// TwinCAT 3 PLC project Machine_Control
// ProgramVersion: 3.1.4024.0
// libraries:
//   Tc2_Drive, * (Beckhoff Automation GmbH)
//   Tc2_EtherCAT, * (Beckhoff Automation GmbH)
//   Tc2_Standard, * (Beckhoff Automation GmbH)
//   Tc2_System, * (Beckhoff Automation GmbH)
//   Tc3_Module, * (Beckhoff Automation GmbH)
// project tree:
//   GVLs/ GVL_Exceptions.TcGVL, GVL_STRUCT.TcGVL, GVL_VAR.TcGVL
//   / PlcTask.TcTTO
//   POUs/ F_SaveExceptionCode.TcPOU, Motors_Speed_IO.TcPOU, Motor_Speed_PID.TcPOU, Safeties_Product_Feed.TcPOU, SpeedControl_SIM.TcPOU, MAIN.TcPOU
// real-time tasks:
//   TASK PlcTask: cycle T#10ms, priority 20, ADS port 350
// I/O:
//   DEVICE Device 1 (EtherCAT Simulation), AmsNetId 192.168.0.15.2.1

CONFIGURATION Machine_Control
    RESOURCE PLC ON TwinCAT3
        TASK PlcTask(INTERVAL := T#10ms, PRIORITY := 20);
        PROGRAM MAIN WITH PlcTask : MAIN;
    END_RESOURCE
END_CONFIGURATION

// ---- GVLs/GVL_Exceptions.TcGVL
{attribute 'qualified_only'}
VAR_GLOBAL CONSTANT
	
	cMaxExc : UINT := 10;	

END_VAR

VAR_GLOBAL
	
	nExcIndex : UINT;
	aExceptionHistory : ARRAY[0..cMaxExc] OF __SYSTEM.ExceptionCode;

END_VAR

// ---- GVLs/GVL_STRUCT.TcGVL
{attribute 'qualified_only'}
VAR_GLOBAL

END_VAR

TYPE 
ST_DriveRef 	:
STRUCT
	
	sNetId		: T_AmsNetId;
	nSlaveAddr	: UINT	:= GVL_VAR.uiSlaveAddr;
	nDriveNo 	: BYTE	:= GVL_VAR.nDriveNum;
	nDriveType	: BYTE	:= GVL_VAR.nDriveType;
	
END_STRUCT
END_TYPE

// ---- GVLs/GVL_VAR.TcGVL
{attribute 'qualified_only'}
VAR_GLOBAL
	
	//integer variables
	//The values of the rotary encoders are stored into these variables
	diMotorEncoder1 	 	: INT;
	diMotorEncoder2 	 	: INT;
	diMotorEncoder3 	 	: INT;
	diMotorEncoder4 	 	: INT;
	
	//Setting the PPR of the encoders used
	iEncoderPPR 			: INT;
	
	//Speed is calculated after each scan of encoder bits and stored into these variables
	//The values are initialized in order to give the UI something to work with after immediate bootup
	diEncoder1ProdSpeed  	: INT := 0;
	diEncoder2ProdSpeed  	: INT := 0;
	diEncoder3ProdSpeed  	: INT := 0;
	diEncoder4ProdSpeed  	: INT := 0;
	
	//The global speed of motors and overall set-speed
	iMotor1GlobalSpeed   	: INT := 0;
	iMotor2GlobalSpeed   	: INT := 0;
	iMotor3GlobalSpeed   	: INT := 0;
	iMotor4GlobalSpeed   	: INT := 0;
	iSetGlobalSpeed      	: INT := 0;
	iGlobalMinimumFaultSpeed: INT := 40; // This value will be user defined
	
	//An hysteresis is important in order to allow micoradjustments in terms of tolerance
	//The values are initialized in order to give the UI something to work with after immediate bootup
	diEncoder1Hysteresis 	: INT := 0;
	diEncoder2Hysteresis 	: INT := 0;
	diEncoder3Hysteresis 	: INT := 0;
	diEncoder4Hysteresis 	: INT := 0;
	
	//Temperature of gluepot/optical in raw data if anaolgue is used 0-4028 depending on the resolution
	//The values are initialized in order to give the UI something to work with after immediate bootup
	iGlueTemperatureRaw  	: INT := 0;
	iRawBoardOptic1 	 	: INT := 0;
	iRawBoardOptic2  	 	: INT := 0;
	iRawBoardOptic3  	 	: INT := 0;
	iRawBoardOptic4 	 	: INT := 0;
	
	//Amount of times a motor's speed has undergone rectification
	
	iMotor1Rect				: INT;
	iMotor2Rect 			: INT;
	iMotor3Rect 			: INT;
	iMotor4Rect 			: INT;
	
	//Program cutt-off distances
	//This keeps track of material distances if motors lose sync of their speed parameters
	//This will be referenced in conjunction with the "Product Ready" flag which must be set BEFORE product is fed
	//Yet IF product is fed, the precondition must remain true; 
	fProductRun : REAL;
	
	//Motor References VIA EtherCAT Comms methodology
	uiSlaveAddr : UINT;
	nDriveNum	: BYTE;
	nDriveType	: BYTE;
	
	
	//boolean variables
	//As far as feasible the booleans will be initialized
	bStartButton 		 	: BOOL := FALSE;
	bStopButton 		 	: BOOL := FALSE;
	bPauseButton 		 	: BOOL := FALSE;
	//System parameters from the main OS/UI
	bSysParamExec 		 	: BOOL := FALSE;
	bSysParamHold 		 	: BOOL := FALSE;
	bSysParamReset 		 	: BOOL := FALSE;
	bSysParam1 			 	: BOOL := FALSE;
	bSysParam2 			 	: BOOL := FALSE;
	//Some IO information about the motor's state
	bMotor1Running 		 	: BOOL := FALSE;
	bMotor2Running 		 	: BOOL := FALSE;
	bMotor3Running 		 	: BOOL := FALSE;
	bMotor4Running 		 	: BOOL := FALSE;
	//Gluepot Boolean indicators
	bGlueReady 			 	: BOOL := FALSE;
	
	//Output Section for controlling the COILS with boolean values
	bStartMotor1			: BOOL := FALSE;
	bStartMotor2			: BOOL := FALSE;
	bStartMotor3			: BOOL := FALSE;
	bStartMotor4			: BOOL := FALSE;
	bMotorsHaveStarted		: BOOL := FALSE;
	
	//Bolleans for controlling the carious motor's speed:
	//These variables are called again in the PID controller POU Motor_Speed_PID
	bIncreaseSpeed1 		: BOOL := FALSE;
	bDecreaseSpeed1 		: BOOL := FALSE;
	bIncreaseSpeed2 		: BOOL := FALSE;
	bDecreaseSpeed2 		: BOOL := FALSE;
	bIncreaseSpeed3 		: BOOL := FALSE;
	bDecreaseSpeed3 		: BOOL := FALSE;
	bIncreaseSpeed4 		: BOOL := FALSE;
	bDecreaseSpeed4 		: BOOL := FALSE;

//Real variables
	//Temperature of glue pot in degrees celsius
	//The values are initialized in order to give the UI something to work with after immediate bootup
	fGlueTemperature 	 	: REAL := 0.0;
	fBoardOptic1 		 	: REAL := 0.0;
	fBoardOptic2 		 	: REAL := 0.0;
	fBoardOptic3 		 	: REAL := 0.0;
	fBoardOptic4 		 	: REAL := 0.0;
	fMaterialDistanceMeter 	: REAL := 0.0;
	fMotor1Thermal 			: REAL := 0.0;
	fMotor2Thermal 			: REAL := 0.0;
	fMotor3Thermal 			: REAL := 0.0;
	fMotor4Thermal 			: REAL := 0.0;
	
	//REAL values for adjusting the motor speeds after having gone through the Motor_Speed_PID POU
	fMotor1AdjustFactor 	: REAL;
	fMotor2AdjustFactor 	: REAL;
	fMotor3AdjustFactor 	: REAL;
	fMotor4AdjustFactor 	: REAL;
	//REAL value for the hysteresis of the motors speed reference provided to the drives from the Motor_Speed_PID POU
	fMotor1Hysteresis		: REAL;
	fMotor2Hysteresis		: REAL;
	fMotor3Hysteresis		: REAL;
	fMotor4Hysteresis		: REAL;
	
	//This is where the parameters for checking the material highs and lows will be stored
	fParametersOptic1 : REAL;
	fParametersOptic2 : REAL;
	fParametersOptic3 : REAL;
	fParametersOptic4 : REAL;
	
END_VAR

// ---- POUs/MAIN.TcPOU
PROGRAM MAIN
VAR
	bSwitchCtrl		: BOOL := TRUE;
	nRotateUpper	: WORD := 16#8000;
	nRotateLower	: WORD := 16#01;
	
	//Variables for dynamically changing the devices spoken to over EtherCAT
	uiSlaveAddr : UINT;
	nDriveNum	: BYTE;
	nDriveType	: BYTE;
	//For the sake of demonstration I am going to employ a CASE switch for talking to the various drives when initializing...
	iNumDrives	: UINT := 1;
	iDriveType	: UINT := 123;
	
	//Hardware inputs
	bEL1004_CH4 AT%I*	: BOOL;
	stPlcDriveRef AT %I* : ST_PlcDriveRef;
	
	
	nEL2008_value AT%Q*	: BYTE;
	bInit1 : BOOL := FALSE;
	bInit2 : BOOL := FALSE;
	bInit3 : BOOL := FALSE;
	bInit4 : BOOL := FALSE;
	
	//Function Block references
	fbWriteCommandControl 	: FB_SoEWriteCommandControl_ByDriveRef;
	bWriteCommand			: BOOL;	
END_VAR

VAR_INPUT
	//Reference to the drive. The reference to the drive can be linked directly to the PLC in the System Manager. 
	//To do this, an instance of the structure ST_PlcDriveRef must be allocated and the NetID must be converted from the byte array into a string. (Type: ST_DriveRef)
	stDriveRef	: ST_DriveRef;
	//Parameter number to which fbWriteCommandControl refers, e.g. "P_0_IDN + 23" for P-0-0023
	nIdn		: WORD;
	//Indicates, if a command should be prepared (eSoE_CmdControl_Set := 1), executed (eSoE_CmdControl_SetAndEnable := 3) or aborted (eSoE_CmdControl_Cancel := 0).
	eCmdControl	: E_SoE_CmdControl;
	//The function block is enabled via a positive edge at this input
	bExecute	: BOOL;
	//Maximum time (10 s) allowed for the execution of the function block.
	tTimeout	: TIME := DEFAULT_ADS_TIMEOUT;	
END_VAR

VAR_OUTPUT
	//This output is set when the function block is activated, and remains set until a feedback is received.
	bBusy			: BOOL;
	//This output is set after the bBusy output has been reset when an error occurs in the transmission of the command.
	bError			: BOOL;
	//In the case of a set bError output returns the ADS error code of the last executed command.
	iAdsErrId		: UINT;
	//In the case of a set bError output returns the Sercos error of the last executed command.
	iSercosErrId	: UINT;
END_VAR

(*This portion is for dynamic drive communication*)

(*Drives have to be made contact with initially before anything can continue...*)

// A __TRY __CATCH __FINALLY clause will be added for exception handling shortly...

CASE iNumDrives OF //probably the conditional control function I like the most...
//Setting up comms for the motion control needs
	1:	IF NOT bInit1 THEN
		
		//change the Slave address
		uiSlaveAddr := iNumDrives;
		GVL_VAR.uiSlaveAddr := uiSlaveAddr;
		//The structure created for the ST_DriveRef expects a Byte format...hence the conversion of the ints...
		GVL_VAR.nDriveNum	:= INT_TO_BYTE(iNumDrives);
		GVL_VAR.nDriveType	:= INT_TO_BYTE(iDriveType);

		stDriveRef.sNetId		:=	F_CreateAmsNetId(stPlcDriveRef.aNetId);
		//The following values have been preconfigured by the FB
		stDriveRef.nSlaveAddr	:=	GVL_VAR.uiSlaveAddr;
		stDriveRef.nDriveNo		:=	GVL_VAR.nDriveNum;
		stDriveRef.nDriveType	:=	GVL_VAR.nDriveType;
	
		IF (stDriveRef.sNetId <> '') AND (stDriveRef.nSlaveAddr <> 0) THEN
		
		bInit1 := TRUE;//initialization completed
		
		END_IF
	
		END_IF
		
		IF bWriteCommand AND bInit1 THEN
	
			fbWriteCommandControl(
				stDriveRef	:= stDriveRef,
				bExecute	:= TRUE,
				tTimeout	:= DEFAULT_ADS_TIMEOUT,
				nIdn		:= P_0_IDN + 23,
				eCmdControl := eCmdControl
				);
		IF NOT	fbWriteCommandControl.bBusy THEN
			fbWriteCommandControl(stDriveRef := stDriveRef, bExecute := FALSE);
			bWriteCommand := FALSE;			
		END_IF
		
		END_IF
		//increment for the next case...
		iNumDrives := iNumDrives + 1;
		
	2:	IF NOT bInit2 THEN
	
		//change the Slave address
		uiSlaveAddr := iNumDrives;
		GVL_VAR.uiSlaveAddr := uiSlaveAddr;
		//The structure created for the ST_DriveRef expects a Byte format...hence the conversion of the ints...
		GVL_VAR.nDriveNum	:= INT_TO_BYTE(iNumDrives);
		GVL_VAR.nDriveType	:= INT_TO_BYTE(iDriveType);

		stDriveRef.sNetId		:=	F_CreateAmsNetId(stPlcDriveRef.aNetId);
		//The following values have been preconfigured by the FB
		stDriveRef.nSlaveAddr	:=	GVL_VAR.uiSlaveAddr;
		stDriveRef.nDriveNo		:=	GVL_VAR.nDriveNum;
		stDriveRef.nDriveType	:=	GVL_VAR.nDriveType;
	
		IF (stDriveRef.sNetId <> '') AND (stDriveRef.nSlaveAddr <> 0) THEN
		
		bInit2 := TRUE;//initialization completed
		
		END_IF
	
		END_IF
		
		IF bWriteCommand AND bInit2 THEN
	
			fbWriteCommandControl(
				stDriveRef	:= stDriveRef,
				bExecute	:= TRUE,
				tTimeout	:= DEFAULT_ADS_TIMEOUT,
				nIdn		:= P_0_IDN + 23,
				eCmdControl := eCmdControl
				);
		IF NOT	fbWriteCommandControl.bBusy THEN
			fbWriteCommandControl(stDriveRef := stDriveRef, bExecute := FALSE);
			bWriteCommand := FALSE;			
		END_IF
		
		END_IF
		//increment for the next case...
		iNumDrives := iNumDrives + 1;
		
		
	
	3:	IF NOT bInit3 THEN
	
		//change the Slave address
		uiSlaveAddr := iNumDrives;
		GVL_VAR.uiSlaveAddr := uiSlaveAddr;
		//The structure created for the ST_DriveRef expects a Byte format...hence the conversion of the ints...
		GVL_VAR.nDriveNum	:= INT_TO_BYTE(iNumDrives);
		GVL_VAR.nDriveType	:= INT_TO_BYTE(iDriveType);

		stDriveRef.sNetId		:=	F_CreateAmsNetId(stPlcDriveRef.aNetId);
		//The following values have been preconfigured by the FB
		stDriveRef.nSlaveAddr	:=	GVL_VAR.uiSlaveAddr;
		stDriveRef.nDriveNo		:=	GVL_VAR.nDriveNum;
		stDriveRef.nDriveType	:=	GVL_VAR.nDriveType;
	
		IF (stDriveRef.sNetId <> '') AND (stDriveRef.nSlaveAddr <> 0) THEN
		
		bInit3 := TRUE;//initialization completed
		
		END_IF
	
		END_IF
		
		IF bWriteCommand AND bInit3 THEN
	
			fbWriteCommandControl(
				stDriveRef	:= stDriveRef,
				bExecute	:= TRUE,
				tTimeout	:= DEFAULT_ADS_TIMEOUT,
				nIdn		:= P_0_IDN + 23,
				eCmdControl := eCmdControl
				);
		IF NOT	fbWriteCommandControl.bBusy THEN
			fbWriteCommandControl(stDriveRef := stDriveRef, bExecute := FALSE);
			bWriteCommand := FALSE;			
		END_IF
		
		END_IF
		//increment for the next case...
		iNumDrives := iNumDrives + 1;
	
	4:	IF NOT bInit4 THEN
	
		//change the Slave address
		uiSlaveAddr := iNumDrives;
		GVL_VAR.uiSlaveAddr := uiSlaveAddr;
		//The structure created for the ST_DriveRef expects a Byte format...hence the conversion of the ints...
		GVL_VAR.nDriveNum	:= INT_TO_BYTE(iNumDrives);
		GVL_VAR.nDriveType	:= INT_TO_BYTE(iDriveType);

		stDriveRef.sNetId		:=	F_CreateAmsNetId(stPlcDriveRef.aNetId);
		//The following values have been preconfigured by the FB
		stDriveRef.nSlaveAddr	:=	GVL_VAR.uiSlaveAddr;
		stDriveRef.nDriveNo		:=	GVL_VAR.nDriveNum;
		stDriveRef.nDriveType	:=	GVL_VAR.nDriveType;
	
		IF (stDriveRef.sNetId <> '') AND (stDriveRef.nSlaveAddr <> 0) THEN
		
		bInit4 := TRUE;//initialization completed
		
		END_IF
	
		END_IF
		
		IF bWriteCommand AND bInit4 THEN
	
			fbWriteCommandControl(
				stDriveRef	:= stDriveRef,
				bExecute	:= TRUE,
				tTimeout	:= DEFAULT_ADS_TIMEOUT,
				nIdn		:= P_0_IDN + 23,
				eCmdControl := eCmdControl
				);
		IF NOT	fbWriteCommandControl.bBusy THEN
			fbWriteCommandControl(stDriveRef := stDriveRef, bExecute := FALSE);
			bWriteCommand := FALSE;			
		END_IF
		
		END_IF
		//increment for the next case...
		iNumDrives := iNumDrives + 1;
END_CASE




IF bEL1004_CH4 THEN
	IF bSwitchCtrl THEN
		bSwitchCtrl := FALSE;
		nRotateLower := ROL(nRotateUpper, 2);
		nRotateUpper := ROR(nRotateUpper, 2);
		nEL2008_value := WORD_TO_BYTE(nRotateLower OR nRotateUpper);
	END_IF
ELSE
		IF NOT bSwitchCtrl THEN
			bSwitchCtrl := TRUE;
		END_IF
END_IF

END_PROGRAM

// ---- POUs/Motor_Speed_PID.TcPOU
PROGRAM Motor_Speed_PID
VAR
	//Global Variables Assignments
	//Increase or decrease the speed depending on the booleans set by the SpeedControl POU
	//The entire existance of this instance of code assumes no common reference of speed 
	//Basically no servo-motors with trusted speeds are used in the process...
	bIncreaseSpeed1 : BOOL := GVL_VAR.bIncreaseSpeed1;
	bDecreaseSpeed1 : BOOL := GVL_VAR.bDecreaseSpeed1;
	bIncreaseSpeed2 : BOOL := GVL_VAR.bIncreaseSpeed2;
	bDecreaseSpeed2 : BOOL := GVL_VAR.bDecreaseSpeed2;
	bIncreaseSpeed3 : BOOL := GVL_VAR.bIncreaseSpeed3;
	bDecreaseSpeed3 : BOOL := GVL_VAR.bDecreaseSpeed3;
	bIncreaseSpeed4 : BOOL := GVL_VAR.bIncreaseSpeed4;
	bDecreaseSpeed4 : BOOL := GVL_VAR.bDecreaseSpeed4;
	
	//The motor VFD controls have to be referenced here as well... This may be done via some etherCAT comms
	
	//Global speed setting for hte reference of the PID
	iSetGlobalSpeed : INT := GVL_VAR.iSetGlobalSpeed;
	fKp : REAL := 0; //Controller amplification, this is the value sent to the motor controller
	//These are the outputs of the Proportional function to be sent to the drives after encoder references.
	fMotor1AdjustFactor : REAL := GVL_VAR.fMotor1AdjustFactor;
	fMotor2AdjustFactor : REAL := GVL_VAR.fMotor2AdjustFactor;
	fMotor3AdjustFactor : REAL := GVL_VAR.fMotor3AdjustFactor;
	fMotor4AdjustFactor : REAL := GVL_VAR.fMotor4AdjustFactor;
	
	//Reference for the varioous drives' addresses
	//Reference to the drive. The reference to the drive can be linked directly to the PLC in the System Manager.
	//To do this, an instance of the structure ST_PlcDriveRef must be allocated and the 
	//NetID must be converted from the byte array into a string
	
	
END_VAR

//Only allow the activation of the speed control segment of the program if the motors have actually started:

WHILE GVL_VAR.bMotorsHaveStarted DO
	
	//Run through the scans to verify whether or not the logic must start:
	IF bIncreaseSpeed1 OR bDecreaseSpeed1 THEN
	
															//This clause is to keep the motors from going in reverse
		IF GVL_VAR.iMotor1GlobalSpeed < iSetGlobalSpeed AND GVL_VAR.iMotor1GlobalSpeed > 0.0 THEN
		//increase the speed and after making sure the speed doesn't exceed the global set variable for the overall speed
		//determine the factor by which the speed should be increased
		
		//The formula for Proportional control is: P = Kp * (Setpoint - Feedback)
		//Or in this case: GVL_VAR.iMotor1GlobalSpeed := fKp * (GVL_VAR.iSetGlobalSpeed - GVl_VAR.iMotor1GlobalSpeed);
		//So it will look like this (remember this automatically returns a REAL number (Fractional/Decimal)):
		//If you wish to turn a REAL value into an INT value: INT_Value := TRUNC(REAL_Value);
		fMotor1AdjustFactor := fKp * (iSetGlobalSpeed - GVL_VAR.iMotor1GlobalSpeed);	
		//Remember to include a function for keeping the hysteresis in mind.
		GVL_VAR.fMotor1AdjustFactor := fMotor1AdjustFactor - GVL_VAR.fMotor1Hysteresis;
		//increase the speed and after making sure the speed doesn't exceed the global set variable for the overall speed


	
		//Reset the booleans responsible for activating this function
		GVL_VAR.bDecreaseSpeed1 := FALSE;
		GVL_VAR.bIncreaseSpeed1 := FALSE;
		ELSE
		//post a speed reference error
		//Reset the booleans responsible for activating this function
		GVL_VAR.bDecreaseSpeed1 := FALSE;
		GVL_VAR.bIncreaseSpeed1 := FALSE;			
		 
			
		END_IF
		
	END_IF
	
		//Run through the scans to verify whether or not the logic must start:
	IF bIncreaseSpeed2 OR bDecreaseSpeed2 THEN
	
		
		IF GVL_VAR.iMotor1GlobalSpeed < iSetGlobalSpeed AND GVL_VAR.iMotor2GlobalSpeed > 0.0 THEN
		fMotor2AdjustFactor := fKp * (iSetGlobalSpeed - GVL_VAR.iMotor2GlobalSpeed);
		GVL_VAR.fMotor2AdjustFactor := fMotor2AdjustFactor - GVL_VAR.fMotor2Hysteresis;
		//increase the speed and after making sure the speed doesn't exceed the global set variable for the overall speed	
		//Reset the booleans responsible for activating this function
		GVL_VAR.bDecreaseSpeed2 := FALSE;
		GVL_VAR.bIncreaseSpeed2 := FALSE;
		ELSE
		//post a speed reference error
		//Reset the booleans responsible for activating this function
		GVL_VAR.bDecreaseSpeed2 := FALSE;
		GVL_VAR.bIncreaseSpeed2 := FALSE;
		END_IF
		
	END_IF
	
		//Run through the scans to verify whether or not the logic must start:
	IF bIncreaseSpeed3 OR bDecreaseSpeed3 THEN
	
		
		IF GVL_VAR.iMotor1GlobalSpeed < iSetGlobalSpeed AND GVL_VAR.iMotor3GlobalSpeed > 0.0 THEN
		fMotor3AdjustFactor := fKp * (iSetGlobalSpeed - GVL_VAR.iMotor3GlobalSpeed);
		GVL_VAR.fMotor3AdjustFactor := fMotor3AdjustFactor - GVL_VAR.fMotor3Hysteresis;
		//increase the speed and after making sure the speed doesn't exceed the global set variable for the overall speed	
		//Reset the booleans responsible for activating this function
		GVL_VAR.bDecreaseSpeed3 := FALSE;
		GVL_VAR.bIncreaseSpeed3 := FALSE;
		ELSE//post a speed reference error
		//Reset the booleans responsible for activating this function
		GVL_VAR.bDecreaseSpeed3 := FALSE;
		GVL_VAR.bIncreaseSpeed3 := FALSE;
		END_IF
		
	END_IF
	
		//Run through the scans to verify whether or not the logic must start:
	IF bIncreaseSpeed4 OR bDecreaseSpeed4 THEN
	
		
		IF GVL_VAR.iMotor1GlobalSpeed < iSetGlobalSpeed AND GVL_VAR.iMotor4GlobalSpeed > 0.0 THEN
		fMotor4AdjustFactor := fKp * (iSetGlobalSpeed - GVL_VAR.iMotor4GlobalSpeed);
		GVL_VAR.fMotor4AdjustFactor := fMotor4AdjustFactor - GVL_VAR.fMotor4Hysteresis;
		//increase the speed and after making sure the speed doesn't exceed the global set variable for the overall speed	
		//Reset the booleans responsible for activating this function
		GVL_VAR.bDecreaseSpeed4 := FALSE;
		GVL_VAR.bIncreaseSpeed4 := FALSE;
		ELSE//post a speed reference error
		//Reset the booleans responsible for activating this function
		GVL_VAR.bDecreaseSpeed4 := FALSE;
		GVL_VAR.bIncreaseSpeed4 := FALSE;
		END_IF
		
	END_IF
	

END_WHILE

END_PROGRAM

// ---- POUs/F_SaveExceptionCode.TcPOU
FUNCTION F_SaveExceptionCode
VAR_INPUT
	excInput : __SYSTEM.ExceptionCode;
END_VAR

IF GVL_Exceptions.nExcIndex <= GVL_Exceptions.cMaxExc THEN
    GVL_Exceptions.aExceptionHistory[GVL_Exceptions.nExcIndex] := excInput;
    GVL_Exceptions.nExcIndex := GVL_Exceptions.nExcIndex + 1;
END_IF

END_FUNCTION

// ---- POUs/Motors_Speed_IO.TcPOU
PROGRAM Motors_Speed_IO
VAR_OUTPUT
	//Values to send to the motors
	fToSend1 : REAL;
	fToSend2 : REAL;
	fToSend3 : REAL;
	fToSend4 : REAL;
	
	//Booleans confirming that something has been sent...
	bSend1Ready : BOOL := FALSE;
	bSend2Ready : BOOL := FALSE;
	bSend3Ready : BOOL := FALSE;
	bSend4Ready : BOOL := FALSE;
END_VAR

VAR
	R_TRIG_0: R_TRIG;
	R_TRIG_1: R_TRIG;
	R_TRIG_2: R_TRIG;
	R_TRIG_3: R_TRIG;
END_VAR
VAR // added by the converter: edge detectors and wires of the graphical bodies
    _w1, _w2, _w3, _w4 : BOOL;
END_VAR

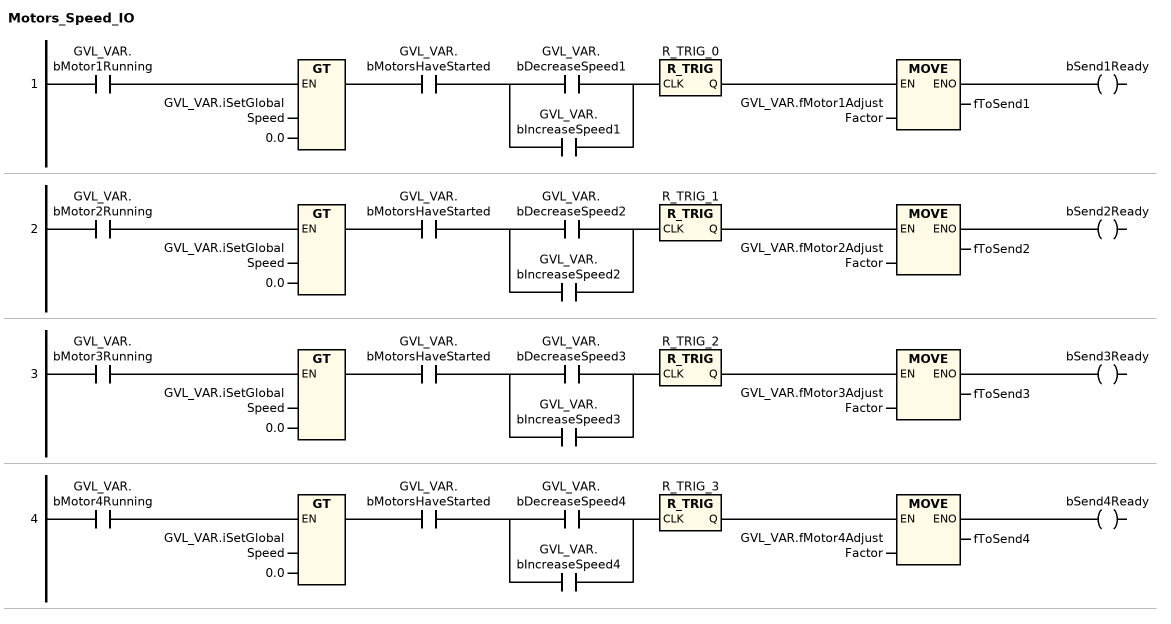
// NETWORK 1
R_TRIG_0(CLK := (GVL_VAR.bMotor1Running AND GVL_VAR.iSetGlobalSpeed > 0.0) AND GVL_VAR.bMotorsHaveStarted AND (GVL_VAR.bDecreaseSpeed1 OR GVL_VAR.bIncreaseSpeed1)); // R_TRIG
_w1 := R_TRIG_0.Q;
IF _w1 THEN fToSend1 := GVL_VAR.fMotor1AdjustFactor; END_IF
bSend1Ready := _w1;

// NETWORK 2
R_TRIG_1(CLK := (GVL_VAR.bMotor2Running AND GVL_VAR.iSetGlobalSpeed > 0.0) AND GVL_VAR.bMotorsHaveStarted AND (GVL_VAR.bDecreaseSpeed2 OR GVL_VAR.bIncreaseSpeed2)); // R_TRIG
_w2 := R_TRIG_1.Q;
IF _w2 THEN fToSend2 := GVL_VAR.fMotor2AdjustFactor; END_IF
bSend2Ready := _w2;

// NETWORK 3
R_TRIG_2(CLK := (GVL_VAR.bMotor3Running AND GVL_VAR.iSetGlobalSpeed > 0.0) AND GVL_VAR.bMotorsHaveStarted AND (GVL_VAR.bDecreaseSpeed3 OR GVL_VAR.bIncreaseSpeed3)); // R_TRIG
_w3 := R_TRIG_2.Q;
IF _w3 THEN fToSend3 := GVL_VAR.fMotor3AdjustFactor; END_IF
bSend3Ready := _w3;

// NETWORK 4
R_TRIG_3(CLK := (GVL_VAR.bMotor4Running AND GVL_VAR.iSetGlobalSpeed > 0.0) AND GVL_VAR.bMotorsHaveStarted AND (GVL_VAR.bDecreaseSpeed4 OR GVL_VAR.bIncreaseSpeed4)); // R_TRIG
_w4 := R_TRIG_3.Q;
IF _w4 THEN fToSend4 := GVL_VAR.fMotor4AdjustFactor; END_IF
bSend4Ready := _w4;

END_PROGRAM

// ---- POUs/Safeties_Product_Feed.TcPOU
PROGRAM Safeties_Product_Feed
VAR_INPUT

	//These will be initialized up until the program has confirmed that these safeties aren't triggered.
	//This also serves as an IO test procedure...
	bPhysicalSafetyFence1 : BOOL;
	bPhysicalSafetyFence2 : BOOL;
	bPhysicalSafetyFence3 : BOOL;
	bPhysicalSafetyFence4 : BOOL;
	bFenceNotCompromised     : BOOL;
	//The proximity sensor responsible for checking if material is indeed present.
	bMaterialPresent : BOOL;
	//This is for the ADSLOGSTR to output a message to the user
	msgCtrlMask  : DWORD;
    msgFmtStr    : T_MaxString;
    strArg       : T_MaxString;

END_VAR

VAR
	
	bSafetiesStartup : BOOL := FALSE;
	//This is a real number for storing the value representin the length of product that has run...
	fProductRun : REAL := GVL_VAR.fProductRun;
	//These are sensors for checking the hight of the product being processed...
	//If they become TRUE, THEN there is a production flow malfunction in terms of the raw material.
	//They are also initialized to TRUE UNTIL proven functional.
	bOpticSensor1 : BOOL := TRUE;
	bOpticSensor2 : BOOL := TRUE;
	bOpticSensor3 : BOOL := TRUE;
	bOpticSensor4 : BOOL := TRUE;
	bProductFlowCompromised : BOOL := TRUE;
	bFieldCommsOK : BOOL := FALSE;

	//Real variables
	//Temperature of glue pot in degrees celsius
	//The values are initialized in order to give the UI something to work with after immediate bootup
	fGlueTemperature 	 	: REAL := GVL_VAR.fGlueTemperature;
	fBoardOptic1 		 	: REAL := GVL_VAR.fBoardOptic1;
	fBoardOptic2 		 	: REAL := GVL_VAR.fBoardOptic2;
	fBoardOptic3 		 	: REAL := GVL_VAR.fBoardOptic3;
	fBoardOptic4 		 	: REAL := GVL_VAR.fBoardOptic4;

	//The REAL values of the motor's thermal characteristics can be obtained via EtherCAT comms.
	fMotor1Thermal 			: REAL := GVL_VAR.fMotor1Thermal;
	fMotor2Thermal 			: REAL := GVL_VAR.fMotor2Thermal;
	fMotor3Thermal 			: REAL := GVL_VAR.fMotor3Thermal;
	fMotor4Thermal 			: REAL := GVL_VAR.fMotor4Thermal;
	
	//This is where the parameters for checking the material highs and lows will be stored
	fParametersOptic1 : REAL := GVL_VAR.fParametersOptic1;
	fParametersOptic2 : REAL := GVL_VAR.fParametersOptic2;
	fParametersOptic3 : REAL := GVL_VAR.fParametersOptic3;
	fParametersOptic4 : REAL := GVL_VAR.fParametersOptic4;
	
	//Allowed variance of material
	//This variable is for storing the allowed fluctiations of material movement...
	fMaterialMinimum1 : REAL;
	fMaterialMinimum2 : REAL;
	fMaterialMinimum3 : REAL;
	fMaterialMinimum4 : REAL;
	
	fMaterialMaximum1 : REAL;
	fMaterialMaximum2 : REAL;
	fMaterialMaximum3 : REAL;
	fMaterialMaximum4 : REAL;
	
	//More ADSLOGSTR variable declarations
	sDefectiveDevice : STRING;
	strSFCErrorStep : STRING; (* Declaration*)
    rtMessageOutput: R_TRIG;
    bSFCError: BOOL;
	udiAdsLogRes: DINT;
	
	cTryCond: INT;
	
	//Variables For the TRY exception Handler
	nCounter1          : INT;
    nCounter2          : INT;
    nCounter_TRY1      : INT;
    nCounter_TRY2      : INT;
    nCounter_CATCH     : INT;    
    nCounter_FINALLY   : INT;
 
    exc                : __SYSTEM.ExceptionCode;
    lastExc            : __SYSTEM.ExceptionCode;
 
    pSample            : POINTER TO BOOL;
    bVar               : BOOL;
    nSample            : INT := 100;
    nDivisor           : INT;
END_VAR

// If any of the safeties are triggered the operator MUST be prompted to a manual reset of the alarm condition.

WHILE NOT bSafetiesStartup DO
	//A TRUE value should be returned.
	bFenceNotCompromised := NOT bPhysicalSafetyFence1 AND NOT bPhysicalSafetyFence2 AND NOT bPhysicalSafetyFence3 AND NOT bPhysicalSafetyFence4;
__TRY
//make contact with all of the EtherCAT devices to ensure proper comms to the devices is established
//Initiate contact 
		
//If contact is successful =>
		bFieldCommsOK := TRUE;
__CATCH(exc);
		//if some sort of error does occur, it should be caught and returned
			rtMessageOutput(CLK := bSFCError);
		IF rtMessageOutput.Q THEN
    		udiAdsLogRes := ADSLOGSTR( msgCtrlMask := ADSLOG_MSGTYPE_ERROR OR ADSLOG_MSGTYPE_MSGBOX,
			 msgFmtStr := 'PLC Msg.: Field Devices Communication Failure At The' + sDefectiveDevice + '%s',
			 strArg := strSFCErrorStep);
			 
			// Exception logging
    		lastExc := exc;
    		F_SaveExceptionCode(excInput := exc);
    		// Correct the faulty variable values
    		IF (exc = __SYSTEM.ExceptionCode.RTSEXCPT_ACCESS_VIOLATION) AND (pSample = 0) THEN
        		pSample  := ADR(bVar);
 			ELSIF ((exc = __SYSTEM.ExceptionCode.RTSEXCPT_DIVIDEBYZERO) OR (exc = __SYSTEM.ExceptionCode.RTSEXCPT_FPU_DIVIDEBYZERO)) AND (nDivisor = 0) THEN
        		nDivisor := 1;
    		END_IF
	
		END_IF;

__FINALLY
		//Else if all is well, send the first values to the end-nodes and receive the first values
		//SAve the state of the communication status into the responsible booleans
		//Return the global variables...
		
__ENDTRY;

	

END_WHILE

WHILE bSafetiesStartup AND bMaterialPresent DO
	
//These instances return a boolean value... If TRUE is returned then all is well...
//Should a FALSE be returned under any circumstances, THEN a "Product jammed" error must be logged
//The sensors should be analogue in nature so as to return a formattible value. The formatted value would be somewhere in the mm range
 
	bOpticSensor1 := fParametersOptic1 < fMaterialMaximum1 AND fParametersOptic1 > fMaterialMinimum1;
	bOpticSensor2 := fParametersOptic2 < fMaterialMaximum2 AND fParametersOptic2 > fMaterialMinimum2;
	bOpticSensor3 := fParametersOptic3 < fMaterialMaximum3 AND fParametersOptic3 > fMaterialMinimum3;
	bOpticSensor4 := fParametersOptic4 < fMaterialMaximum4 AND fParametersOptic4 > fMaterialMinimum4;

END_WHILE

END_PROGRAM

// ---- POUs/SpeedControl_SIM.TcPOU
PROGRAM SpeedControl_SIM
VAR
	
//Boolean values for determining the speed at which the motors are running in a controlled and called fashion.
	bEncCallMade1   	: BOOL := FALSE;
	bEncCallMade2   	: BOOL := FALSE;
	bEncCallMade3   	: BOOL := FALSE;
	bEncCallMade4   	: BOOL := FALSE;
	bMotor1Running  	: BOOL := GVL_VAR.bMotor1Running;
	bMotor2Running  	: BOOL := GVL_VAR.bMotor2Running;
	bMotor3Running  	: BOOL := GVL_VAR.bMotor3Running;
	bMotor4Running  	: BOOL := GVL_VAR.bMotor4Running;
	bProgramStarted 	: BOOL := GVL_VAR.bStartButton;
	bMotorsHaveStarted  : BOOL := GVL_VAR.bMotorsHaveStarted;
	bFirstReading		: BOOL;
	bSpeedCheck1Pass	: BOOL;
	bSpeedCheck2Pass	: BOOL;
	bSpeedCheck3Pass	: BOOL;
	bSpeedCheck4Pass	: BOOL;
	
//Global Variables into which the encoder values will be stored.
	iEncoder1Val 		: INT := GVL_VAR.diMotorEncoder1;
	iEncoder2Val 		: INT := GVL_VAR.diMotorEncoder2;
	iEncoder3Val 		: INT := GVL_VAR.diMotorEncoder3;
	iEncoder4Val 		: INT := GVL_VAR.diMotorEncoder4;
	iEncoderPPR			: INT := GVL_VAR.iEncoderPPR;
	
//Hysteresis of the encoders...
	iEncoder1Hys 		: INT := GVL_VAR.diEncoder1Hysteresis;
	iEncoder2Hys 		: INT := GVL_VAR.diEncoder2Hysteresis;
	iEncoder3Hys 		: INT := GVL_VAR.diEncoder3Hysteresis;
	iEncoder4Hys 		: INT := GVL_VAR.diEncoder4Hysteresis;
	
//Retrieve the speed settings for the scope of the flow and assign them to local variable names...
	iGlobalSpeedSetting : INT := GVL_VAR.iSetGlobalSpeed;
	iMotor1Speed 		: INT := GVL_VAR.iMotor1GlobalSpeed;
	iMotor2Speed 		: INT := GVL_VAR.iMotor2GlobalSpeed;
	iMotor3Speed 		: INT := GVL_VAR.iMotor3GlobalSpeed;
	iMotor4Speed 		: INT := GVL_VAR.iMotor4GlobalSpeed;
	
//This is primarily used for storing the encoder values and comparisons between motor speeds...
	iMotor1SpeedA		: INT := 0;
	iMotor2SpeedA		: INT := 0;
	iMotor3SpeedA		: INT := 0;
	iMotor4SpeedA		: INT := 0;
	
//Timer functions for controlling the encoder value polling
	tEncCallMadeTimer 	: TON;
	timerDone 			: BOOL := FALSE;
END_VAR

(*Simulated Program*)
//This is for determining the speed of the motors and displaying it on the UI. It is also
// responsible for making sure that all of the motors are indeed running the same speed through measurement.
//This measurement is then taken and it adjusts the speed of the motors accordingly (just for the sake of testing the logic of course)
//If after a certain amount of adjustments the speed still seems unbalanced, THEN the machine will switch off the motor controls and flag a product JAM.
//Give the command to start the motors

IF bProgramStarted THEN
	GVL_VAR.bStartMotor1 := TRUE;
	GVL_VAR.bStartMotor2 := TRUE;
	GVL_VAR.bStartMotor3 := TRUE;
	GVL_VAR.bStartMotor4 := TRUE;
ELSE 
	GVL_VAR.bStartMotor1 := FALSE;
	GVL_VAR.bStartMotor2 := FALSE;
	GVL_VAR.bStartMotor3 := FALSE;
	GVL_VAR.bStartMotor4 := FALSE;
END_IF

//Confirm whether or not the motors have started...
IF bMotor1Running AND bMotor2Running AND bMotor3Running AND bMotor4Running THEN
	//Set the global variable GVL_VAR.bMotorsHaveStarted to TRUE if ALL of the run feedback signals are TRUE
	GVL_VAR.bMotorsHaveStarted := TRUE;
ELSE
	//Set the global variable GVL_VAR.bMotorsHaveStarted to FALSE if NOT ALL of the run feedback signals are TRUE
	GVL_VAR.bMotorsHaveStarted := FALSE;
END_IF

WHILE bMotorsHaveStarted DO 
	//Start the timer for orderky data calls
	IF NOT timerDone THEN
		tEncCallMadeTimer(IN := TRUE, PT:=T#100MS, Q=> timerDone);
	
		IF NOT bEncCallMade1 AND tEncCallMadeTimer.ET = T#25MS  THEN
			iMotor1Speed := iEncoder1Val - iEncoder1Hys;
			iMotor1SpeedA := iEncoder1Val;
			//ensure that the process isn't executed every single new scan cycle by using a boolean trigger
			bEncCallMade1 := TRUE;
			//now the iMotor1Speed Can be formatted and made available to the UI
		END_IF
		
		IF NOT bEncCallMade2 AND tEncCallMadeTimer.ET = T#50MS  THEN
			iMotor2Speed := iEncoder2Val - iEncoder3Hys;
			iMotor2SpeedA := iEncoder2Val;
			//ensure that the process isn't executed every single new scan cycle by using a boolean trigger
			bEncCallMade2 := TRUE;
			//now the iMotor2Speed Can be formatted and made available to the UI
		END_IF
	
		IF NOT bEncCallMade3 AND tEncCallMadeTimer.ET = T#75MS  THEN
			iMotor3Speed := iEncoder3Val - iEncoder3Hys;
			iMotor3SpeedA := iEncoder3Val;
			//ensure that the process isn't executed every single new scan cycle by using a boolean trigger
			bEncCallMade3 := TRUE;
			//now the iMotor3Speed Can be formatted and made available to the UI
		END_IF
	
		IF NOT bEncCallMade4 AND tEncCallMadeTimer.ET = T#100MS  THEN
			iMotor4Speed := iEncoder4Val - iEncoder4Hys;
			iMotor4SpeedA := iEncoder4Val;
			//ensure that the process isn't executed every single new scan cycle by using a boolean trigger
			bEncCallMade4 := TRUE;
			//now the iMotor4Speed Can be formatted and made available to the UI
		END_IF

		IF timerDone AND bEncCallMade4 THEN
			bEncCallMade1 := FALSE;
			bEncCallMade2 := FALSE;
			bEncCallMade3 := FALSE;
			bEncCallMade4 := FALSE;
			tEncCallMadeTimer.IN := FALSE;
			tEncCallMadeTimer.Q := FALSE;
			bFirstReading := TRUE;
			
		END_IF
	END_IF


	
END_WHILE
//Reference in essense a PID controller for all of these motors
//Compare all of the motor's speeds with the main speed setting
WHILE bFirstReading DO
	
	IF iMotor1Speed = iGlobalSpeedSetting THEN
		bSpeedCheck1Pass := TRUE;
		GVL_VAR.bIncreaseSpeed1 := FALSE;
		GVL_VAR.bDecreaseSpeed1 := FALSE;
	ELSE IF iMotor1Speed > iGlobalSpeedSetting THEN
			//DECREASE motor speed!
			bSpeedCheck1Pass := FALSE;
			GVL_VAR.bDecreaseSpeed1 := TRUE;
			
		ELSE //INCREASE motor speed!
			bSpeedCheck1Pass := FALSE;
			GVL_VAR.bIncreaseSpeed1 := TRUE;
		END_IF
	END_IF
	
	IF iMotor2Speed = iGlobalSpeedSetting THEN
		bSpeedCheck2Pass := TRUE;
		GVL_VAR.bIncreaseSpeed2 := FALSE;
		GVL_VAR.bDecreaseSpeed2 := FALSE;

	ELSE IF iMotor2Speed > iGlobalSpeedSetting THEN
		//DECREASE motor speed!
		bSpeedCheck2Pass := FALSE;
		GVL_VAR.bDecreaseSpeed2 := TRUE;
		
		ELSE //INCREASE motor speed!
			bSpeedCheck2Pass := FALSE;
			GVL_VAR.bIncreaseSpeed2 := TRUE;
		END_IF
	END_IF
	
	IF iMotor3Speed = iGlobalSpeedSetting THEN
		bSpeedCheck3Pass := TRUE;
		GVL_VAR.bIncreaseSpeed3 := FALSE;
		GVL_VAR.bDecreaseSpeed3 := FALSE;
	
	ELSE IF iMotor3Speed > iGlobalSpeedSetting THEN
		//DECREASE motor speed!
		bSpeedCheck3Pass := FALSE;
		GVL_VAR.bDecreaseSpeed3 := TRUE;
		
		ELSE //INCREASE motor speed!
			bSpeedCheck3Pass := FALSE;
			GVL_VAR.bIncreaseSpeed3 := TRUE;
		END_IF
	
	END_IF
	
	
	IF iMotor4Speed = iGlobalSpeedSetting THEN
		bSpeedCheck4Pass := TRUE;
		GVL_VAR.bIncreaseSpeed4 := FALSE;
		GVL_VAR.bDecreaseSpeed4 := FALSE;
		
	ELSE IF iMotor4Speed > iGlobalSpeedSetting THEN
		//DECREASE motor speed!
		bSpeedCheck4Pass := FALSE;
		GVL_VAR.bDecreaseSpeed4 := TRUE;
		
		ELSE //INCREASE motor speed!
			bSpeedCheck4Pass := FALSE;
			GVL_VAR.bIncreaseSpeed4 := TRUE;
		END_IF
	
	END_IF

	
END_WHILE

END_PROGRAM
